Universal Robots PolyScope program: p2 joan.urp

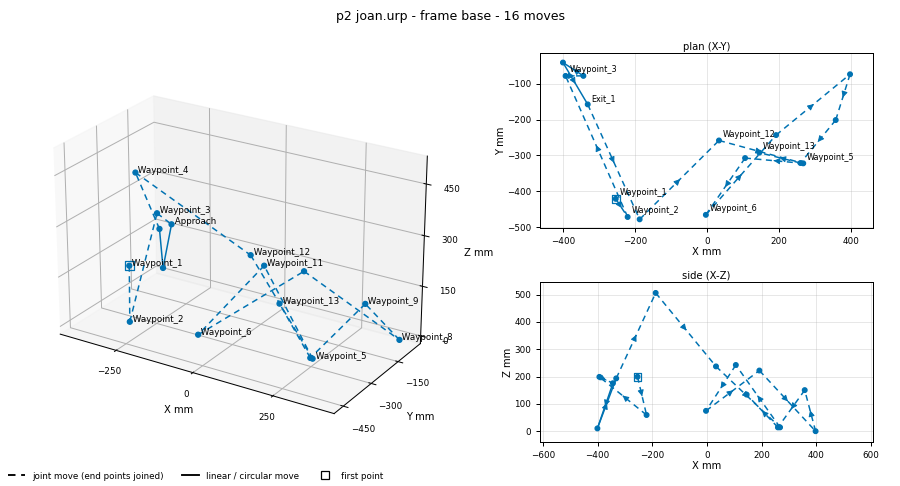
[picture p0: tool path of p2 joan.urp in frame base, 16 of 16 moves have a stored position in this frame; points joined in program order, loops and branches not executed]
Program p2 joan (installation=default directory=/programs createdIn=5.14.5 lastSavedIn=5.14.5 robotSerialNumber=20195300809)
Calibrated DH parameters: a=[-0.000085, -0.20076, -0.212369, 0.000121, -0.000118, 0]; d=[0.15185, -26.306375, 24.753047, 1.684739, 0.085386, 0.092088]; alpha=[1.572149, -0.00522, -0.011864, 1.571339, -1.571085, 0]; deltaTheta=[0, 0.599885, -0.513355, -0.086555, 0.000006, 0]
InitVariablesNode variables(variable(name=Pallet_1_cnt_1, expression=1), variable(name=Pallet_1_lct, expression=1), variable(name=Pallet_1_lno, expression=1), variable(name=Pallet_1_sep, expression=False), variable(name=Pallet_1_tct, expression=1))
Robot Program (runOnlyOnce=false)
  URCap Gripper Activate (Robotiq_Grippers, Robotiq Inc.) dataModel(ResetAndActivateKey=false)
  MoveJ speed 60 deg/s, acceleration 80 deg/s^2 (useActiveTCP=true) feature=Base
    Waypoint Waypoint_1: TCP in base x=-254.411 y=-420.519 z=199.426 mm, rx=0.1943 ry=3.0617 rz=-0.4984 rad; joints [34.363, -61.06, 41.867, -80.946, -75.238, -46.858] deg; TCP offset x=0 y=0 z=174 mm, rx=0 ry=0 rz=0 rad
    MoveJ speed 60 deg/s, acceleration 80 deg/s^2 (useActiveTCP=true) feature=Base
      Waypoint Waypoint_2: TCP in base x=-221.3 y=-470.922 z=59.608 mm, rx=-0.0493 ry=3.0866 rz=-0.1111 rad; joints [47.563, -36.529, 29.89, -84.306, -85.883, -44.239] deg
    URCap Gripper (Robotiq_Grippers, Robotiq Inc.) dataModel(position=49.01960784313725, force=0.0, speed=0.0, positionInDouble=49.01960784313725, forceInDouble=0.0, speedInDouble=0.0, slaveIds=[9], blocking=true)
    MoveJ speed 60 deg/s, acceleration 80 deg/s^2 (useActiveTCP=true) feature=Base
      Waypoint Waypoint_3: TCP in base x=-393.857 y=-78.761 z=198.992 mm, rx=-2.0087 ry=-2.0662 rz=0.3366 rad; joints [-10.182, -90.958, 83.945, -101.879, -87.601, -11.286] deg
      URCap Palletizing (polyscope-pallet-impl, Universal Robots) dataModel(palletFeature=Base, isPalletizing=true, Variable(key=referencePoint, variable(featureName=referencePoint)), Variable(key=separatorPoint, variable(featureName=separatorPoint)), Variable(key=name, variable(name=Pallet_1)), Variable(key=globalCountingVariable, variable(name=Pallet_1_cnt_1, initializeExpression=1)), Variable(key=layerNumberVariable, variable(name=Pallet_1_lno, initializeExpression=1)), Variable(key=layerCountingVariable, variable(name=Pallet_1_lct, initializeExpression=1)), Variable(key=handleSeparatorVariable, variable(name=Pallet_1_sep, initializeExpression=False)), Variable(key=totalCountVariable, variable(name=Pallet_1_tct, initializeExpression=1)), Length(key=objectHeight value=0.02 unit=M)); state(isChildrenLocked=true)
        URCap Patterns (polyscope-pallet-impl, Universal Robots) state(isChildrenLocked=true)
          URCap Pattern (polyscope-pallet-impl, Universal Robots) dataModel(UUID=60f2ebae-c33d-4eb8-9f0c-d9da8bc98b41, patternType=GRID, rows=3, columns=2, Variable(key=nameVariable, variable(name=Grid_Pattern_1))); state(isChildrenLocked=true)
            URCap Item (polyscope-pallet-impl, Universal Robots) dataModel(UUID=88dc2b69-a6a0-407f-a235-212e3f587432, patternType=GRID, index=0, calibrationDeltaTheta=[2.0871938292282843E-8, 0.5998849625986696, -0.513354759222901, -0.08655474087847535, 6.239817607139875E-6, -6.658617090343766E-8], calibrationA=[-8.52060452638757E-5, -0.2007601879611388, -0.2123691625519033, 1.2105607098011576E-4, -1.1833705743435544E-4, 0.0], calibrationD=[0.15184970286177432, -26.306374840159272, 24.75304670983349, 1.6847390881089916, 0.085385969004481, 0.09208826337351553], calibrationAlpha=[1.5721487795181908, -0.005219907129425837, -0.011864150755780208, 1.5713392161993658, -1.5710853432049288, 0.0], calibrationJointChecksum=[-1860213401, -1859864814, -1494669377, -1328152407, -1329437658, -1329056899], calibrationStatus=2, calibrationValidChecksum=true, baseToFeature=[0.0, 0.0, 0.0, 0.0, 0.0, 0.0], TCPOffset=[1.0945518896424145E-5, -2.4416600208687633E-5, 0.17399055198133778, 4.7075802821076185E-5, 9.958452709144454E-6, 7.564399619092801E-5], Variable(key=variable, variable(name=CornerItem_1)), JointPositions(key=jointpositions, JointPosition(key=[1], Angle(key=pos value=-0.291976 unit=RAD)), JointPosition(key=[2], Angle(key=pos value=-1.342269 unit=RAD)), JointPosition(key=[3], Angle(key=pos value=1.947813 unit=RAD)), JointPosition(key=[4], Angle(key=pos value=-2.276604 unit=RAD)), JointPosition(key=[5], Angle(key=pos value=-1.534619 unit=RAD)), JointPosition(key=[6], Angle(key=pos value=-0.283905 unit=RAD))))
            URCap Item (polyscope-pallet-impl, Universal Robots) dataModel(UUID=76b7c95c-5c52-439a-89b7-da5c97bcced7, patternType=GRID, index=1, calibrationDeltaTheta=[2.0871938292282843E-8, 0.5998849625986696, -0.513354759222901, -0.08655474087847535, 6.239817607139875E-6, -6.658617090343766E-8], calibrationA=[-8.52060452638757E-5, -0.2007601879611388, -0.2123691625519033, 1.2105607098011576E-4, -1.1833705743435544E-4, 0.0], calibrationD=[0.15184970286177432, -26.306374840159272, 24.75304670983349, 1.6847390881089916, 0.085385969004481, 0.09208826337351553], calibrationAlpha=[1.5721487795181908, -0.005219907129425837, -0.011864150755780208, 1.5713392161993658, -1.5710853432049288, 0.0], calibrationJointChecksum=[-1860213401, -1859864814, -1494669377, -1328152407, -1329437658, -1329056899], calibrationStatus=2, calibrationValidChecksum=true, baseToFeature=[0.0, 0.0, 0.0, 0.0, 0.0, 0.0], TCPOffset=[-9.855743570513775E-6, -1.1849120150730919E-5, 0.17398289050311463, 4.2262277702407554E-5, -2.746784874396136E-5, -2.8996802479806453E-5], Variable(key=variable, variable(name=CornerItem_2)), JointPositions(key=jointpositions, JointPosition(key=[1], Angle(key=pos value=0.32867 unit=RAD)), JointPosition(key=[2], Angle(key=pos value=-1.01105 unit=RAD)), JointPosition(key=[3], Angle(key=pos value=1.486434 unit=RAD)), JointPosition(key=[4], Angle(key=pos value=-2.15288 unit=RAD)), JointPosition(key=[5], Angle(key=pos value=-1.66803 unit=RAD)), JointPosition(key=[6], Angle(key=pos value=0.309686 unit=RAD))))
            URCap Item (polyscope-pallet-impl, Universal Robots) dataModel(UUID=f3124642-abb9-4294-8bd3-7ccca49d07e4, patternType=GRID, index=2, calibrationDeltaTheta=[2.0871938292282843E-8, 0.5998849625986696, -0.513354759222901, -0.08655474087847535, 6.239817607139875E-6, -6.658617090343766E-8], calibrationA=[-8.52060452638757E-5, -0.2007601879611388, -0.2123691625519033, 1.2105607098011576E-4, -1.1833705743435544E-4, 0.0], calibrationD=[0.15184970286177432, -26.306374840159272, 24.75304670983349, 1.6847390881089916, 0.085385969004481, 0.09208826337351553], calibrationAlpha=[1.5721487795181908, -0.005219907129425837, -0.011864150755780208, 1.5713392161993658, -1.5710853432049288, 0.0], calibrationJointChecksum=[-1860213401, -1859864814, -1494669377, -1328152407, -1329437658, -1329056899], calibrationStatus=2, calibrationValidChecksum=true, baseToFeature=[0.0, 0.0, 0.0, 0.0, 0.0, 0.0], TCPOffset=[1.076663173654735E-5, -1.4395080566942386E-5, 0.17399831138923244, 2.5639152533134377E-5, -1.8942758788512257E-5, 4.038845339292608E-6], Variable(key=variable, variable(name=CornerItem_3)), JointPositions(key=jointpositions, JointPosition(key=[1], Angle(key=pos value=0.242367 unit=RAD)), JointPosition(key=[2], Angle(key=pos value=-0.598142 unit=RAD)), JointPosition(key=[3], Angle(key=pos value=0.781048 unit=RAD)), JointPosition(key=[4], Angle(key=pos value=-1.986573 unit=RAD)), JointPosition(key=[5], Angle(key=pos value=-1.63565 unit=RAD)), JointPosition(key=[6], Angle(key=pos value=0.230578 unit=RAD))))
            URCap Item (polyscope-pallet-impl, Universal Robots) dataModel(UUID=8fb6b438-cc9d-4f73-87a5-d081fe9542d6, patternType=GRID, index=3, calibrationDeltaTheta=[2.0871938292282843E-8, 0.5998849625986696, -0.513354759222901, -0.08655474087847535, 6.239817607139875E-6, -6.658617090343766E-8], calibrationA=[-8.52060452638757E-5, -0.2007601879611388, -0.2123691625519033, 1.2105607098011576E-4, -1.1833705743435544E-4, 0.0], calibrationD=[0.15184970286177432, -26.306374840159272, 24.75304670983349, 1.6847390881089916, 0.085385969004481, 0.09208826337351553], calibrationAlpha=[1.5721487795181908, -0.005219907129425837, -0.011864150755780208, 1.5713392161993658, -1.5710853432049288, 0.0], calibrationJointChecksum=[-1860213401, -1859864814, -1494669377, -1328152407, -1329437658, -1329056899], calibrationStatus=2, calibrationValidChecksum=true, baseToFeature=[0.0, 0.0, 0.0, 0.0, 0.0, 0.0], TCPOffset=[-1.5450463735186722E-6, 1.0229964896413257E-5, 0.17400558737019167, -3.1855282407429153E-5, -2.1305811642756473E-5, 3.9607091418328144E-5], Variable(key=variable, variable(name=CornerItem_4)), JointPositions(key=jointpositions, JointPosition(key=[1], Angle(key=pos value=-0.181293 unit=RAD)), JointPosition(key=[2], Angle(key=pos value=-0.658333 unit=RAD)), JointPosition(key=[3], Angle(key=pos value=0.771375 unit=RAD)), JointPosition(key=[4], Angle(key=pos value=-1.661112 unit=RAD)), JointPosition(key=[5], Angle(key=pos value=-1.574983 unit=RAD)), JointPosition(key=[6], Angle(key=pos value=-0.269287 unit=RAD))))
        URCap Layers (polyscope-pallet-impl, Universal Robots) dataModel(separators=[false], selectedPatterns=[60f2ebae-c33d-4eb8-9f0c-d9da8bc98b41])
        URCap At Each Item (polyscope-pallet-impl, Universal Robots) dataModel(currentWizardState=MANUAL, selectedPattern=60f2ebae-c33d-4eb8-9f0c-d9da8bc98b41, selectedPosition=88dc2b69-a6a0-407f-a235-212e3f587432, Pose(key=refBaseToFeature, Position(key=posePosition, Length(key=X value=0 unit=M), Length(key=Y value=0 unit=M), Length(key=Z value=0 unit=M)), Rotation(key=poseRotation, Angle(key=RX value=0 unit=RAD), Angle(key=RY value=0 unit=RAD), Angle(key=RZ value=0 unit=RAD))), Pose(key=refPose, Position(key=posePosition, Length(key=X value=-0.369631 unit=M), Length(key=Y value=-0.039678 unit=M), Length(key=Z value=0.012936 unit=M)), Rotation(key=poseRotation, Angle(key=RX value=-2.185587 unit=RAD), Angle(key=RY value=-2.160609 unit=RAD), Angle(key=RZ value=0.137825 unit=RAD))))
          URCap Generated Movements (polyscope-pallet-impl, Universal Robots) state(isChildrenLocked=true)
            MoveJ speed 60 deg/s, acceleration 80 deg/s^2 (useActiveTCP=true) feature=referencePoint
              Waypoint Approach: TCP in base x=-344.357 y=-78.618 z=175.791 mm, rx=-1.9955 ry=-1.9695 rz=0.4215 rad; joints [-13.074, -109.457, 109.297, -113.865, -85.932, -11.399] deg; feature pose in base x=-369.631 y=-39.678 z=12.936 mm, rx=-2.1856 ry=-2.1606 rz=0.1378 rad
            MoveL speed 250 mm/s, acceleration 1200 mm/s^2 (useActiveTCP=true) feature(featureName=referencePoint)
              Waypoint ToolActionPoint: TCP in base x=-401.128 y=-41.591 z=10.524 mm, rx=-2.0906 ry=-2.1179 rz=0.2407 rad; joints [-15.755, -73.567, 112.771, -141.5, -86.833, -16.54] deg
            Folder Tool action
              URCap Gripper (Robotiq_Grippers, Robotiq Inc.) dataModel(position=18.03921568627451, force=0.0, speed=0.0, positionInDouble=18.03921568627451, forceInDouble=0.0, speedInDouble=0.0, slaveIds=[9], blocking=true)
            MoveL speed 250 mm/s, acceleration 1200 mm/s^2 (useActiveTCP=true) feature(featureName=referencePoint)
              Waypoint Exit_1: TCP in base x=-332.295 y=-157.925 z=193.53 mm, rx=-1.8995 ry=-1.8642 rz=0.6774 rad; joints [3.539, -113.487, 118.572, -131.386, -89.532, 4.7] deg
      MoveJ speed 60 deg/s, acceleration 80 deg/s^2 (useActiveTCP=true) feature=Base
        Waypoint Waypoint_4: TCP in base x=-187.956 y=-477.474 z=506.035 mm, rx=-0.0237 ry=-2.204 rz=2.2073 rad; joints [21.411, -82.453, 75.589, -171.453, -23.184, -2.158] deg
      MoveJ speed 60 deg/s, acceleration 80 deg/s^2 (useActiveTCP=true) feature=Base
        Waypoint Waypoint_12: TCP in base x=32.631 y=-258.242 z=237.329 mm, rx=-0.0818 ry=3.0678 rz=-0.5369 rad; joints [46.267, -128.11, 92.694, -67.939, -75.602, -44.534] deg
      MoveJ speed 60 deg/s, acceleration 80 deg/s^2 (useActiveTCP=true) feature=Base
        Waypoint Waypoint_5: TCP in base x=266.887 y=-321.814 z=14.373 mm, rx=0.0457 ry=-3.1196 rz=0.2406 rad; joints [114.056, -66.061, 97.163, -128.987, -94.806, 21.722] deg
        URCap Gripper (Robotiq_Grippers, Robotiq Inc.) dataModel(position=50.19607843137255, force=0.0, speed=0.0, positionInDouble=50.19607843137255, forceInDouble=0.0, speedInDouble=0.0, slaveIds=[9], blocking=true)
      MoveJ speed 60 deg/s, acceleration 80 deg/s^2 (useActiveTCP=true) feature=Base
        Waypoint Waypoint_11: TCP in base x=105.19 y=-307.138 z=242.506 mm, rx=-0.0607 ry=3.0332 rz=-0.6809 rad; joints [78.026, -115.897, 95.094, -93.581, -83.427, -12.527] deg
      MoveJ speed 60 deg/s, acceleration 80 deg/s^2 (useActiveTCP=true) feature=Base
        Waypoint Waypoint_6: TCP in base x=-3.862 y=-464.981 z=74.824 mm, rx=-0.0523 ry=-3.1093 rz=0.2256 rad; joints [72.437, -62.445, 74.263, -110.174, -89.757, -15.766] deg
        URCap Gripper (Robotiq_Grippers, Robotiq Inc.) dataModel(position=0.0, force=0.0, speed=0.0, positionInDouble=0.0, forceInDouble=0.0, speedInDouble=0.0, slaveIds=[9], blocking=true)
      MoveJ speed 60 deg/s, acceleration 80 deg/s^2 (useActiveTCP=true) feature=Base
        Waypoint Waypoint_7: TCP in base x=191.345 y=-243.219 z=222.244 mm, rx=0.0057 ry=-3.1311 rz=0.1994 rad; joints [104.746, -96.948, 74.622, -74.67, -92.825, 14.756] deg
      MoveJ speed 60 deg/s, acceleration 80 deg/s^2 (useActiveTCP=true) feature=Base
        Waypoint Waypoint_8: TCP in base x=396.956 y=-74.154 z=0.33 mm, rx=-0.0173 ry=-3.1293 rz=0.1919 rad; joints [154.868, -63.08, 94.099, -123.696, -97.244, 65.028] deg
      URCap Gripper (Robotiq_Grippers, Robotiq Inc.) dataModel(position=50.19607843137255, force=0.0, speed=0.0, positionInDouble=50.19607843137255, forceInDouble=0.0, speedInDouble=0.0, slaveIds=[9], blocking=true)
      MoveJ speed 60 deg/s, acceleration 80 deg/s^2 (useActiveTCP=true) feature=Base
        Waypoint Waypoint_9: TCP in base x=357.165 y=-201.453 z=150.574 mm, rx=0.0831 ry=2.9429 rz=-0.7408 rad; joints [144.611, -83.56, 95.265, -123.47, -110.323, 53.753] deg
      MoveJ speed 60 deg/s, acceleration 80 deg/s^2 (useActiveTCP=true) feature=Base
        Waypoint Waypoint_10: TCP in base x=259.219 y=-320.909 z=14.257 mm, rx=0.0656 ry=-3.1123 rz=0.1684 rad; joints [112.709, -65.68, 94.955, -124.576, -94.262, 19.803] deg
        URCap Gripper (Robotiq_Grippers, Robotiq Inc.) dataModel(position=0.0, force=0.0, speed=0.0, positionInDouble=0.0, forceInDouble=0.0, speedInDouble=0.0, slaveIds=[9], blocking=true)
      MoveJ speed 60 deg/s, acceleration 80 deg/s^2 (useActiveTCP=true) feature=Base
        Waypoint Waypoint_13: TCP in base x=144.839 y=-292.073 z=134.269 mm, rx=-0.1038 ry=3.0738 rz=-0.4307 rad; joints [90.141, -107.846, 112.758, -110.808, -88.163, -3.424] deg
Thread Thread_1 (runOnlyOnce=false)
  If digital_in[0] ≟ False
    Set DigitalOutput pin=digital_out[0]; digitalValue=0
  Else 
    Set DigitalOutput pin=digital_out[0]; digitalValue=1
